// TIA Portal V16 export
// export: Created 2024-04-26T21:24:43.8751024Z, ExportSetting WithDefaults, DisplayName Totally Integrated Automation Portal, DisplayVersion V16, DisplayName TIA Portal Version Control Interface, DisplayVersion V16, DisplayName TIA Portal Openness, DisplayVersion V16, DisplayName STEP 7 Professional, DisplayVersion V16, DisplayName STEP 7 Safety, DisplayVersion V16, DisplayName WinCC Professional, DisplayVersion V16
DATA_BLOCK "MC_Home_DB_2"   // DB26
// stored: AutoNumber true, InstanceOfName MC_Home, OfSystemLibElement MC_Home, OfSystemLibVersion 6.0
"MC_Home"
   // VAR_INPUT
   //    Axis : TO_Axis;
   //    Execute : Bool;
   //    Position : Real;
   //    Mode : Int;
   // END_VAR
   // VAR_OUTPUT
   //    Done : Bool;
   //    Busy : Bool;
   //    CommandAborted : Bool;
   //    Error : Bool;
   //    ErrorID : Word;
   //    ErrorInfo : Word;
   //    ReferenceMarkPosition : Real;
   // END_VAR
   // VAR
   //    FB_ID : DInt;
   // END_VAR
BEGIN
END_DATA_BLOCK
